SUBAPPLICATION Softkey_Aux_Auto_IXA_TO_Remote_WRITE (* VT-SoftKey lesen ODER AUX-Zuweisung (Joystick) lesen ODER lokaler Web-Override ODER Automatik-Kommando + Remote-OPC-UA-Write an Zielmodul (generisch, ein Kanal, ohne Status-Feedback). Kopie von Softkey_Aux_IXA_TO_Remote_WRITE + 1 zusaetzlicher AUTO_IN-Socket - fuer Funktionen mit autonomer Ansteuerung (z.B. Achslenkung-Mittelpunkt-Automatik). *)
  (* Standard: 61499-2 *)
  (* Version 1.2, 2026-09-16, Franz Höpfinger, Fix: SUBSCRIBE_WEB.OUT konnte nicht an 2 Ziele (OR_MERGE.IN3 UND WEB_STATE) gleichzeitig angeschlossen werden - Adapter-Plugs sind strikt 1:1, kein Fan-out wie bei Daten-/Eventverbindungen (FORTE-Bootfehler INVALID_STATE beim 2. CREATE Connection auf demselben Plug). AX_SPLIT_2 (SPLIT_WEB) dazwischengesetzt, analog dem bereits etablierten SPLIT_Y/AR_SPLIT_2-Muster. *)
  (* Version 1.1, 2026-09-16, Franz Höpfinger, Neuer Ausgangs-Plug WEB_STATE ergaenzt (reiner Fan-out von SUBSCRIBE_WEB.OUT) - behebt Doppel-Self-Subscribe auf ID_WEB_READ (FORTE: 'Cannot add another one'), da Fahrwerk_Mittelpunkt_Automatik denselben Knoten bisher selbst nochmal abonniert hat. Siehe BERICHT_2026-09-16_STG3_I1_I3_I4_I6_STALE_REMOTE_SUBSCRIBE.md Abschnitt 16-17. *)
  (* Version 1.0, 2026-09-11, Franz Höpfinger, Kopie von Softkey_Aux_IXA_TO_Remote_WRITE (Version 1.0, 2026-09-07) + AUTO_IN-Socket (AX_OR_4 statt AX_OR_3) fuer Achslenkung-Mittelpunkt-Automatik. Nur fuer Kanaele mit Automatik-Bedarf verwenden - alle anderen Verwender von Softkey_Aux_IXA_TO_Remote_WRITE(_BG_OPC) bleiben unveraendert auf dem Original-Typ. *)
  PACKAGE MyLib::sys;
  IMPORT isobus::UT::Q::const::IDs::ID_NULL;
  (* Documentation:
  SoftKey UND Aux UND Automatik → Remote-OPC-UA-Write (nur Kommando, kein Status)
   Kopie von Softkey_Aux_IXA_TO_Remote_WRITE mit einem 4. ODER-Eingang (AUTO_IN, AX_OR_4 statt AX_OR_3) fuer eine autonome Ansteuerung (z.B. Achslenkung-Mittelpunkt-Automatik). Genau EIN Publisher pro Kanal auf ID_WRITE_REMOTE bleibt dadurch erhalten, auch wenn 4 statt 3 Quellen zusammengefuehrt werden - kein Self-Latch-Risiko.
   Kein Status-Feedback/Hintergrundfarbe hier - dafuer AX_SUBSCRIBE_BG3_WEB_OPC danebenstellen (unveraendert, gleiche u16ObjId/u16ObjIdA-Werte durchreichen) - siehe Softkey_Aux_Auto_IXA_TO_Remote_WRITE_BG_OPC fuer die vorverdrahtete Kombination.
   WEB_STATE (neu, Version 1.1): Plug von SUBSCRIBE_WEB.OUT ueber SPLIT_WEB (AX_SPLIT_2) durchgereicht, damit andere Composite-Instanzen (z.B. Fahrwerk_Mittelpunkt_Automatik fuer die Override-Erkennung) denselben Web-Zustand per normaler Adapterverbindung lesen koennen, statt selbst nochmal denselben Knoten lokal zu abonnieren - FORTE erlaubt nur EINEN lokalen OPC-UA-Subscriber pro Knoten. SPLIT_WEB ist noetig, da ein Adapter-Plug (anders als Daten-/Eventverbindungen) nicht an 2 Ziele gleichzeitig angeschlossen werden kann (Version 1.2 Fix, siehe VersionInfo).
  *)
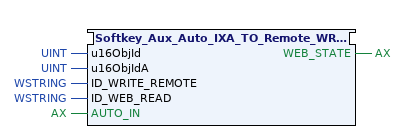
  VAR_INPUT
    u16ObjId : UINT := ID_NULL; (* Object ID SoftKey (VT) *)
    u16ObjIdA : UINT := ID_NULL; (* Object ID AuxFunction2 (VT) *)
    ID_WRITE_REMOTE : WSTRING; (* Remote-Write-Adresse zum Zielmodul (Befehl, ACTION=WRITE, CLIENT) *)
    ID_WEB_READ : WSTRING; (* Lokale Subscribe-Adresse fuer einen Web-Client (z.B. vt-ui-mirror) auf demselben Modul, ODER-verknuepft mit SoftKey und AUX *)
  END_VAR
  SOCKETS
    AUTO_IN : adapter::types::unidirectional::AX; (* Autonomes Kommando (z.B. Achslenkung-Mittelpunkt-Automatik), ODER-verknuepft mit SoftKey/Aux/Web *)
  END_SOCKETS
  PLUGS
    WEB_STATE : adapter::types::unidirectional::AX; (* Web-Zustand (= SUBSCRIBE_WEB.OUT) nach aussen durchgereicht, damit andere Composite-Instanzen denselben Wert per Datenverbindung nutzen koennen statt selbst nochmal lokal zu abonnieren (nur 1 lokaler OPC-UA-Subscriber pro Knoten zulaessig) *)
  END_PLUGS
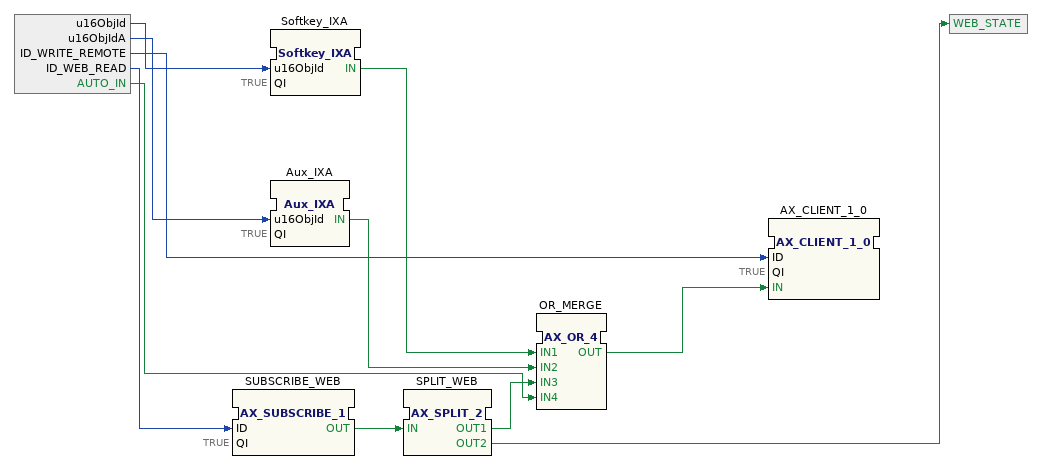
  FBS
    Softkey_IXA : isobus::UT::io::Softkey::Softkey_IXA(QI := TRUE);
    Aux_IXA : isobus::UT::io::Auxiliary::IN::Aux_IXA(QI := TRUE);
    SUBSCRIBE_WEB : adapter::net::AX_SUBSCRIBE_1(QI := TRUE);
    OR_MERGE : adapter::booleanOperators::AX_OR_4;
    SPLIT_WEB : adapter::events::unidirectional::AX_SPLIT_2;
    AX_CLIENT_1_0 : adapter::net::AX_CLIENT_1_0(QI := TRUE);
  END_FBS
  DATA_CONNECTIONS
    u16ObjId TO Softkey_IXA.u16ObjId;
    u16ObjIdA TO Aux_IXA.u16ObjId;
    ID_WEB_READ TO SUBSCRIBE_WEB.ID;
    ID_WRITE_REMOTE TO AX_CLIENT_1_0.ID;
  END_CONNECTIONS
  ADAPTER_CONNECTIONS
    Softkey_IXA.IN TO OR_MERGE.IN1;
    Aux_IXA.IN TO OR_MERGE.IN2;
    SUBSCRIBE_WEB.OUT TO SPLIT_WEB.IN;
    SPLIT_WEB.OUT1 TO OR_MERGE.IN3;
    AUTO_IN TO OR_MERGE.IN4;
    OR_MERGE.OUT TO AX_CLIENT_1_0.IN;
    SPLIT_WEB.OUT2 TO WEB_STATE;
  END_CONNECTIONS
END_SUBAPPLICATION
